Yaskawa INFORM job: UNTITLED.JBI

/JOB
//NAME UNTITLED
///FOLDERNAME INNE
//POS
///NPOS 0,0,0,0,0,0
//INST
///DATE 2023/10/04 15:16
///ATTR SC,RW
///GROUP1 RB1,BS1,ST1
NOP
'UNTITLED
CALL JOB:W3
CALL JOB:W5
CALL JOB:W7
END
